FUNCTION_BLOCK SBActor (* Actor for setting the battery transfer of a Sonnenbatterie in slave mode via its RESTful API *)
  (* Standard: 61499-2; Description: Requires the http communication layer. *)
  (* Version 1.0, 2017-08-27, Marc Jakobi, HTW Berlin *)
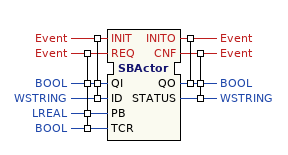
  EVENT_INPUT
    INIT WITH QI, ID; (* Initialization Request *)
    REQ WITH QI, PB, TCR; (* Normal Execution Request *)
  END_EVENT
  EVENT_OUTPUT
    INITO WITH QO; (* Initialization Confirm *)
    CNF WITH QO, STATUS; (* Execution Confirmation *)
  END_EVENT
  VAR_INPUT
    QI : BOOL; (* Input event qualifier *)
    ID : WSTRING; (* Connection identifier (ip:port) *)
    PB : LREAL; (* Battery transfer (positive = charge, negative = discharge) *)
    TCR : BOOL; (* Indicator for trickle charge (true if battery was just released from trickle charge) *)
  END_VAR
  VAR_OUTPUT
    QO : BOOL; (* Output event qualifier *)
    STATUS : WSTRING; (* HTTP responses *)
  END_VAR
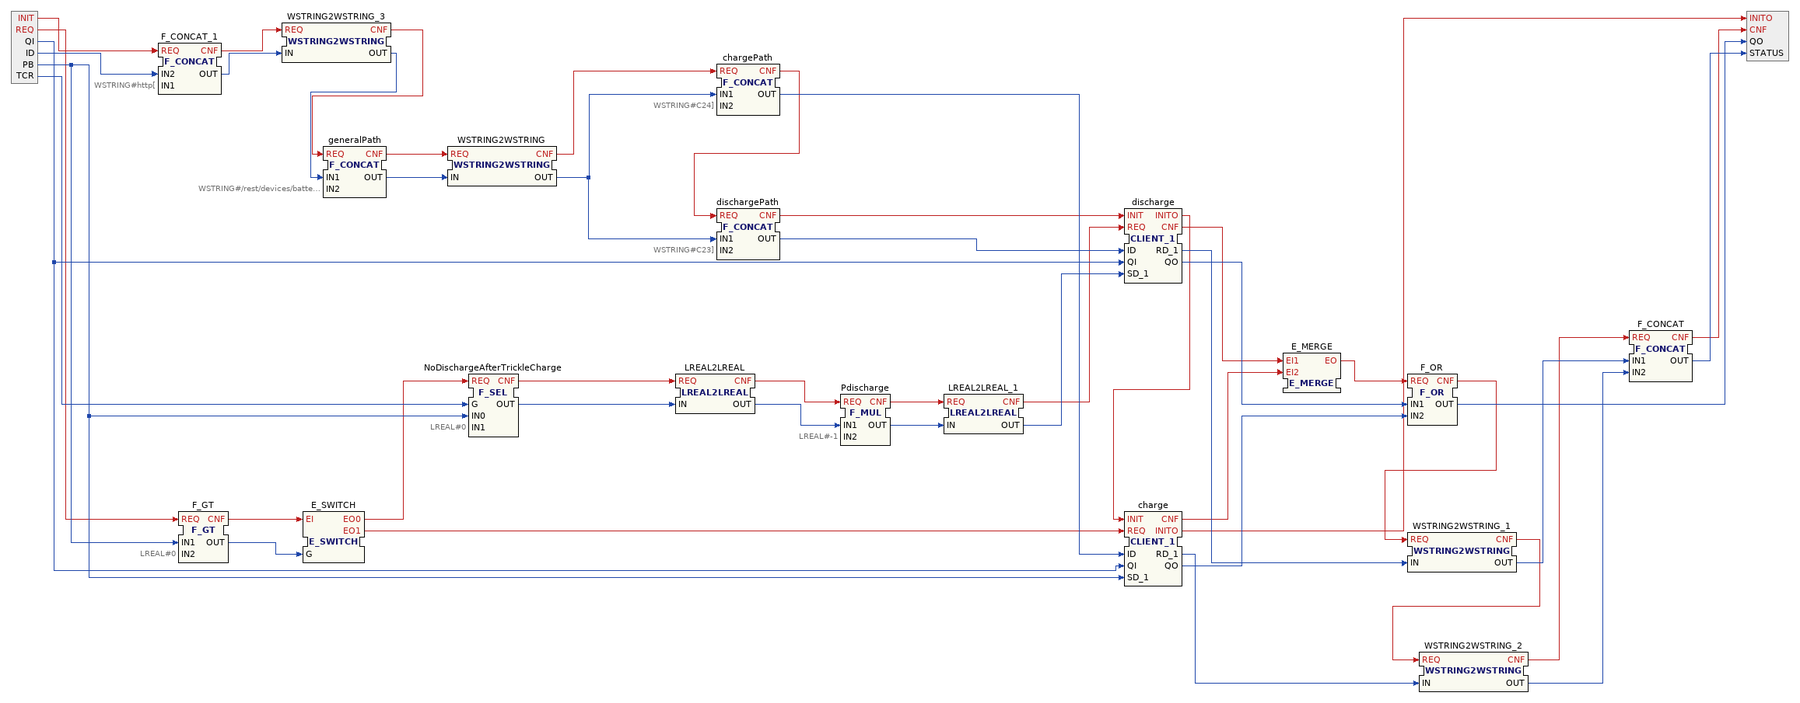
  FBS
    generalPath : F_CONCAT(IN2 := WSTRING#/rest/devices/battery/);
    chargePath : F_CONCAT(IN2 := WSTRING#C24]);
    dischargePath : F_CONCAT(IN2 := WSTRING#C23]);
    WSTRING2WSTRING : WSTRING2WSTRING;
    F_GT : F_GT(IN2 := LREAL#0);
    E_SWITCH : E_SWITCH;
    NoDischargeAfterTrickleCharge : F_SEL(IN1 := LREAL#0);
    Pdischarge : F_MUL(IN2 := LREAL#-1);
    LREAL2LREAL : LREAL2LREAL;
    LREAL2LREAL_1 : LREAL2LREAL;
    discharge : CLIENT_1;
    charge : CLIENT_1;
    E_MERGE : E_MERGE;
    WSTRING2WSTRING_1 : WSTRING2WSTRING;
    WSTRING2WSTRING_2 : WSTRING2WSTRING;
    F_CONCAT : F_CONCAT;
    F_OR : F_OR;
    F_CONCAT_1 : F_CONCAT(IN1 := WSTRING#http[);
    WSTRING2WSTRING_3 : WSTRING2WSTRING;
  END_FBS
  EVENT_CONNECTIONS
    generalPath.CNF TO WSTRING2WSTRING.REQ;
    WSTRING2WSTRING.CNF TO chargePath.REQ;
    chargePath.CNF TO dischargePath.REQ;
    REQ TO F_GT.REQ;
    F_GT.CNF TO E_SWITCH.EI;
    E_SWITCH.EO0 TO NoDischargeAfterTrickleCharge.REQ;
    NoDischargeAfterTrickleCharge.CNF TO LREAL2LREAL.REQ;
    LREAL2LREAL.CNF TO Pdischarge.REQ;
    Pdischarge.CNF TO LREAL2LREAL_1.REQ;
    dischargePath.CNF TO discharge.INIT;
    LREAL2LREAL_1.CNF TO discharge.REQ;
    discharge.INITO TO charge.INIT;
    E_SWITCH.EO1 TO charge.REQ;
    discharge.CNF TO E_MERGE.EI1;
    charge.CNF TO E_MERGE.EI2;
    WSTRING2WSTRING_1.CNF TO WSTRING2WSTRING_2.REQ;
    WSTRING2WSTRING_2.CNF TO F_CONCAT.REQ;
    F_CONCAT.CNF TO CNF;
    charge.INITO TO INITO;
    E_MERGE.EO TO F_OR.REQ;
    F_OR.CNF TO WSTRING2WSTRING_1.REQ;
    INIT TO F_CONCAT_1.REQ;
    F_CONCAT_1.CNF TO WSTRING2WSTRING_3.REQ;
    WSTRING2WSTRING_3.CNF TO generalPath.REQ;
  END_CONNECTIONS
  DATA_CONNECTIONS
    generalPath.OUT TO WSTRING2WSTRING.IN;
    WSTRING2WSTRING.OUT TO chargePath.IN1;
    WSTRING2WSTRING.OUT TO dischargePath.IN1;
    PB TO F_GT.IN1;
    F_GT.OUT TO E_SWITCH.G;
    TCR TO NoDischargeAfterTrickleCharge.G;
    PB TO NoDischargeAfterTrickleCharge.IN0;
    NoDischargeAfterTrickleCharge.OUT TO LREAL2LREAL.IN;
    LREAL2LREAL.OUT TO Pdischarge.IN1;
    Pdischarge.OUT TO LREAL2LREAL_1.IN;
    dischargePath.OUT TO discharge.ID;
    QI TO discharge.QI;
    LREAL2LREAL_1.OUT TO discharge.SD_1;
    chargePath.OUT TO charge.ID;
    QI TO charge.QI;
    PB TO charge.SD_1;
    discharge.RD_1 TO WSTRING2WSTRING_1.IN;
    charge.RD_1 TO WSTRING2WSTRING_2.IN;
    WSTRING2WSTRING_1.OUT TO F_CONCAT.IN1;
    WSTRING2WSTRING_2.OUT TO F_CONCAT.IN2;
    F_CONCAT.OUT TO STATUS;
    discharge.QO TO F_OR.IN1;
    charge.QO TO F_OR.IN2;
    F_OR.OUT TO QO;
    ID TO F_CONCAT_1.IN2;
    F_CONCAT_1.OUT TO WSTRING2WSTRING_3.IN;
    WSTRING2WSTRING_3.OUT TO generalPath.IN1;
  END_CONNECTIONS
END_FUNCTION_BLOCK
